TYPE ST_ProductStats  :
STRUCT
   averageWeight : REAL;
   minWeight     : REAL;
   maxWeight     : REAL;
   defectiveCount: INT;
END_STRUCT
END_TYPE

(* stored: Version 1.1.0.1, ProductVersion 3.1.4024.16
   DUT ST_ProductStats: Id {a76e0c6f-8a7d-4ca2-96d7-9b5400e0ab85} *)
